# B&R Automation Studio project Test
Automation Studio 3.0.90.20 SP02; Default project

## Configuration Simulation

### Task classes (Cpu.sw)
```
Cyclic#4:
  NewProgram <- NewProgram.prg
Libraries: AsIecCon, astime
```

## Logical view

### Global.typ - Global data types
```iecst
(********************************************************************
 * COPYRIGHT --
 ********************************************************************
 * File: Global.typ
 * Author: anton
 * Created: December 11, 2013
 ********************************************************************
 * Global data types of project test
 ********************************************************************)

TYPE
	gOPCType : 	STRUCT
		Input : StructInput;
		Output : StructOutput;
	END_STRUCT;
END_TYPE

(*gOPC.Output*)

TYPE
	StructOutput : 	STRUCT
		Xpos : REAL;
		Ypos : REAL;
		Zpos : REAL;
		load : BOOL;
		DI : BOOL;
		DOutput : BOOL;
		status : UINT;
		drivestatus : UINT;
		driveack : BOOL;
		ack : BOOL;
	END_STRUCT;
END_TYPE

(*gOPC.Input*)

TYPE
	StructInput : 	STRUCT
		start : BOOL;
		src_cell : USINT;
		dst_cell : USINT;
		command : USINT;
	END_STRUCT;
END_TYPE
```

### Global.var - Global variables
```iecst
(********************************************************************
 * COPYRIGHT --
 ********************************************************************
 * File: Global.var
 * Author: anton
 * Created: December 11, 2013
 ********************************************************************
 * Global variables of project test
 ********************************************************************)
VAR
	gOPC : gOPCType := (0);
END_VAR
```

### Program Logical/NewProgram (ANSIC) - A new program

#### NewProgram.c - Implementation code
```c
/********************************************************************
 * COPYRIGHT --
 ********************************************************************
 * Program: NewProgram
 * File: NewProgram.c
 * Author: anton
 * Created: December 11, 2013
 ********************************************************************
 * Implementation of program NewProgram
 ********************************************************************/

#include <bur/plctypes.h>

#ifdef _DEFAULT_INCLUDES
	#include <AsDefault.h>
#endif

void _INIT NewProgramINIT(void)
{
	/* TODO: Add code here */
	gOPC.Input.command=0;
	gOPC.Input.dst_cell=0;
	gOPC.Input.src_cell=0;
	gOPC.Input.start=0;

	gOPC.Output.ack=0;
	gOPC.Output.DI=0;
	gOPC.Output.DOutput=0;
	gOPC.Output.driveack=0;
	gOPC.Output.drivestatus=0;
	gOPC.Output.load=0;
	gOPC.Output.status=0;
	gOPC.Output.Xpos=0;
	gOPC.Output.Ypos=0;
	gOPC.Output.Zpos=0;
}

void _CYCLIC NewProgramCYCLIC(void)
{
	/* TODO: Add code here */
	gOPC.Output.Xpos = gOPC.Output.Xpos+0.1;
	if(gOPC.Output.Xpos>200) gOPC.Output.Xpos=0;

}
```

Listed in the project but not available here: Logical/Libraries
